// TwinCAT 3 PLC project benchmark
// ProgramVersion: 3.1.4026.13
// libraries:
//   Struckig, * (Stefan Besler)
//   Tc2_Standard, * (Beckhoff Automation GmbH)
//   Tc2_System, * (Beckhoff Automation GmbH)
//   Tc2_Utilities, * (Beckhoff Automation GmbH)
//   Tc3_Module, * (Beckhoff Automation GmbH)
// project tree:
//   / PlcTask.TcTTO
//   POUs/ MAIN.TcPOU
//   POUs/MovingStatistic/ MovingStatistic.TcPOU
//   POUs/Randomizer/ Randomizer.TcPOU
//   POUs/Random/ IRandom.TcIO, RandomGaussian.TcPOU, RandomUniform.TcPOU
//   POUs/Random/_Test/ RandomGaussianTest.TcPOU
// real-time tasks:
//   TASK PlcTask: cycle T#1ms, priority 1, ADS port 350

CONFIGURATION benchmark
    RESOURCE PLC ON TwinCAT3
        TASK PlcTask(INTERVAL := T#1ms, PRIORITY := 1);
        PROGRAM MAIN WITH PlcTask : MAIN;
    END_RESOURCE
END_CONFIGURATION

// ---- POUs/Random/IRandom.TcIO
INTERFACE IRandom

/// Returns the next random variable
METHOD Next : LREAL
END_METHOD

METHOD SetSeed
VAR_INPUT
  seed : INT;
END_VAR
END_METHOD

END_INTERFACE

// ---- POUs/MAIN.TcPOU
PROGRAM MAIN
VAR CONSTANT
  Dofs : ARRAY [0..3] OF SINT := [1, 3, 6, 7];
  IterationCount : INT := 5;
  TrajactoryCount : DINT := 64 * 1024;
END_VAR
VAR
  _positionDist : RandomGaussian(seed:=42, mu:=0, sigma:=4);
  _dynamicDist : RandomGaussian(seed:=43, mu:=0, sigma:=0.8);
  _limitDist : RandomUniform(seed:=44, lowerBound:=0, upperBound:=4);
  
  _p : Randomizer(_positionDist);
  _d : Randomizer(_dynamicDist);
  _l : Randomizer(_limitDist);
  
  _otg : Struckig.Otg(cycletime:=0.001, dofs:=0);
  
  _step : INT := 0;
  _dt, _it, _jt : DINT := 0;
  
  _trajectoryStatistic, _itStatistic, _worstStatistic : MovingStatistic;
  
  _averageMean, _worstMean, _averageSigma, _worstSigma : ARRAY[0..3] OF LREAL; 
  
  _cpucounter : Tc2_System.GETCPUACCOUNT;
END_VAR

REPEAT
  CASE _step
  OF
    // setup ****************************************************
    0: 
    // **********************************************************

      _otg.FB_init(TRUE, TRUE, 0.001, dofs:=Dofs[_dt]);
      _trajectoryStatistic.Reset();
      _itStatistic.Reset();
      _worstStatistic.Reset();
      
      _p.Fill(ADR(_otg.CurrentPosition), Dofs[_dt]);
      _p.Fill(ADR(_otg.TargetPosition), Dofs[_dt]);
      _l.FillMax(ADR(_otg.maxVelocity), Dofs[_dt], ADR(_otg.TargetVelocity));
      _l.FillMax(ADR(_otg.maxAcceleration), Dofs[_dt], ADR(_otg.TargetAcceleration));
      _l.Fill(ADR(_otg.maxJerk), Dofs[_dt]);
      CheckCalculation(_otg);  
    
      _step := 1;
  
    // iterate start ********************************************
    1: 
    // **********************************************************
    
      _trajectoryStatistic.Reset();
      _step := 2;
      
    // iterate loop *********************************************
    2: 
    // **********************************************************
    
      _p.Fill(ADR(_otg.CurrentPosition), Dofs[_dt]);
      _d.FillOrZero(ADR(_otg.CurrentVelocity), Dofs[_dt], 0.9);
      _d.FillOrZero(ADR(_otg.CurrentAcceleration), Dofs[_dt], 0.8);
      _p.Fill(ADR(_otg.TargetPosition), Dofs[_dt]);
      _d.FillOrZero(ADR(_otg.TargetVelocity), Dofs[_dt], 0.7);
      _d.FillOrZero(ADR(_otg.TargetAcceleration), Dofs[_dt], 0.6);
      _l.FillMax(ADR(_otg.MaxVelocity), Dofs[_dt], ADR(_otg.TargetVelocity));
      _l.FillMax(ADR(_otg.MaxAcceleration), Dofs[_dt], ADR(_otg.TargetAcceleration));
      _l.Fill(ADR(_otg.MaxJerk), Dofs[_dt]);
  
      IF NOT _otg.ValidateInput(FALSE, TRUE)
      THEN
        RETURN;
      END_IF
  
      _trajectoryStatistic.Append(CheckCalculation(_otg));
      _jt := _jt + 1;
      IF _jt > TrajactoryCount
      THEN
        _it := _it + 1;
        _jt := 0;        
        _step := 1;
        _itStatistic.Append(_trajectoryStatistic.Mean);
        _worstStatistic.Append(_trajectoryStatistic.Maximum);
      END_IF
      
      IF _it > IterationCount
      THEN
        _step := 3;
      END_IF
      
    // iterate end **********************************************
    3: 
    // **********************************************************

      _it := 0;
      _jt := 0;
      _averageMean[_dt] := _itStatistic.Mean;
      _averageSigma[_dt] := _itStatistic.Sigma;
      _worstMean[_dt] := _worstStatistic.Mean;
      _worstSigma[_dt] := _worstStatistic.Sigma;      
      _dt := _dt + 1;
      _step := SEL(_dt > 3, 0, 4);

    // done******* **********************************************
    4: 
    // **********************************************************
      ; 
  END_CASE
UNTIL _step = 4 
AND_THEN TRUE // wtf, fix this already Beckhoff - no breakpoints without an additional condition!!!! 
END_REPEAT

_step := 4;

METHOD CheckCalculation : LREAL;
VAR_INPUT
  otg : REFERENCE TO Struckig.Otg;
END_VAR
VAR
  cpuAccount : UDINT;
END_VAR
_cpucounter(cpuAccountDW => cpuAccount);
otg();
_cpucounter();
CheckCalculation := (_cpucounter.cpuAccountDW - cpuAccount) * 0.1; // us
END_METHOD

END_PROGRAM

// ---- POUs/Random/RandomGaussian.TcPOU
FUNCTION_BLOCK RandomGaussian IMPLEMENTS IRandom
VAR
  _mu : LREAL;
  _sigma : LREAL;    
  _rnd : Tc2_System.DRAND;
END_VAR

METHOD FB_init : BOOL
VAR_INPUT
	bInitRetains : BOOL; // if TRUE, the retain variables are initialized (warm start / cold start)
	bInCopyCode : BOOL;  // if TRUE, the instance afterwards gets moved into the copy code (online change)
  seed : INT;  
  mu : LREAL;
  sigma : LREAL;
END_VAR
SetSeed(seed);
SetMean(mu);
SetSigma(sigma);
END_METHOD

/// Implementation of the Box-Muller transform for normal distributed random
/// variables. There are much faster methods for doing this.
/// Implementation taken from [here](https://en.wikipedia.org/wiki/Box%E2%80%93Muller_transform)
METHOD Next : LREAL
VAR
  u1, u2 : LREAL;
END_VAR
VAR CONSTANT
  Pi : LREAL := 3.14159265358979323846;
END_VAR
//create two random numbers, make sure u1 is greater than epsilon
REPEAT
  _rnd(Num => u1);
  _rnd(Num => u2);  
UNTIL u1 > 1E-8 END_REPEAT

//compute z0 and z1
Next  := (_sigma * SQRT(-2.0 * LOG(u1))) * COS(2*Pi * u2) + _mu;

// we do not need the 2nd randomly distributed variable
// z1 := mag * SIN(2*Struckig.Constants.Pi  * u2) + mu;
END_METHOD

METHOD FINAL SetMean
VAR_INPUT
  mu : LREAL;
END_VAR
_mu := mu;
END_METHOD

METHOD FINAL SetSeed
VAR_INPUT
  seed : INT;
END_VAR
_rnd.Seed := seed;
END_METHOD

METHOD FINAL SetSigma
VAR_INPUT
  sigma : LREAL;
END_VAR
_sigma := sigma;
END_METHOD

END_FUNCTION_BLOCK

// ---- POUs/Random/RandomUniform.TcPOU
FUNCTION_BLOCK RandomUniform IMPLEMENTS IRandom
VAR
  _lowerBound : LREAL;
  _upperBound : LREAL;  
  _rnd : Tc2_System.DRAND;
END_VAR

METHOD FB_init : BOOL
VAR_INPUT
	bInitRetains : BOOL; // if TRUE, the retain variables are initialized (warm start / cold start)
	bInCopyCode : BOOL;  // if TRUE, the instance afterwards gets moved into the copy code (online change)
  seed : INT;      
  lowerBound : LREAL;
  upperBound : LREAL;
END_VAR
SetSeed(seed);
SetBounds(lowerBound, upperBound);
END_METHOD

METHOD Next : LREAL
_rnd();
Next := _rnd.Num * (_upperBound-_lowerBound) + _lowerBound;
END_METHOD

METHOD FINAL SetBounds
VAR_INPUT
  lowerBound : LREAL;
  upperBound : LREAL;
END_VAR
_lowerBound := lowerBound;
_upperBound := upperBound;
END_METHOD

METHOD FINAL SetSeed
VAR_INPUT
  seed : INT;
END_VAR
_rnd.Seed := seed;
END_METHOD

END_FUNCTION_BLOCK

// ---- POUs/Randomizer/Randomizer.TcPOU
FUNCTION_BLOCK Randomizer
VAR
  _rndUniform : RandomUniform(seed:=0, lowerBound:=0, upperBound:=1);
  _rnd : IRandom;
END_VAR

METHOD FB_init : BOOL
VAR_INPUT
	bInitRetains : BOOL; // if TRUE, the retain variables are initialized (warm start / cold start)
	bInCopyCode : BOOL;  // if TRUE, the instance afterwards gets moved into the copy code (online change)
  rnd : IRandom;
END_VAR
_rnd := rnd;
END_METHOD

METHOD Fill
VAR_INPUT
  data : POINTER TO LREAL;
  size : INT;
END_VAR
VAR
  i : INT;
END_VAR
FOR i:=0 TO size-1
DO
  data[i] := _rnd.Next();
END_FOR
END_METHOD

METHOD FillMax
VAR_INPUT
  data : POINTER TO LREAL;
  size : INT;
  offset : POINTER TO LREAL;
END_VAR
VAR
  i : INT;
END_VAR
FOR i:=0 TO size-1
DO
  data[i] := _rnd.Next() + ABS(offset[i]);
END_FOR
END_METHOD

METHOD FillMin
VAR_INPUT
  data : POINTER TO LREAL;
  size : INT;
  offset : POINTER TO LREAL;
END_VAR
VAR
  i : INT;
END_VAR
FOR i:=0 TO size-1
DO
  data[i] := _rnd.Next() - ABS(offset[i]);
END_FOR
END_METHOD

METHOD FillOrZero
VAR_INPUT
  data : POINTER TO LREAL;
  size : INT;
  p : LREAL; // value between 0-1 to adjust the probability of "fill with random number" to "fill with zero". p = 0.9 means that 10% of values are filled with zero
END_VAR
VAR
  i : INT;
END_VAR
FOR i:=0 TO size-1
DO
  data[i] := SEL(_rndUniform.Next() < p, 0, _rnd.Next());
END_FOR
END_METHOD

END_FUNCTION_BLOCK

// ---- POUs/MovingStatistic/MovingStatistic.TcPOU
FUNCTION_BLOCK MovingStatistic
VAR_OUTPUT
  Mean : LREAL;
  Sigma : LREAL;
  Size : DINT;
  Maximum : LREAL;
  Minimum : LREAL;
END_VAR
VAR
  _meanMem : LREAL;
  _varianceSum : LREAL;
END_VAR

METHOD Append
VAR_INPUT
  value : LREAL;
END_VAR
Size := Size + 1;
_meanMem := Mean;
Mean := (Mean + (value - Mean) / DINT_TO_LREAL(Size)); 

IF Size > 1
THEN
  _varianceSum := _varianceSum + (value - Mean) * (value - _meanMem);
  Sigma := SQRT(_varianceSum / (DINT_TO_LREAL(Size) - 1.0));
END_IF

IF value < Minimum
THEN
  Minimum := value;
END_IF

IF value > Maximum
THEN
  Maximum := value;
END_IF
END_METHOD

METHOD FB_init : BOOL
VAR_INPUT
	bInitRetains : BOOL; // if TRUE, the retain variables are initialized (warm start / cold start)
	bInCopyCode : BOOL;  // if TRUE, the instance afterwards gets moved into the copy code (online change)
END_VAR
Reset();
END_METHOD

METHOD FINAL Reset
VAR_INPUT
END_VAR
Mean := 0;
Sigma := 0;
Size := 0;
Minimum := 1.7976931348623157E+308;
Maximum := -1.7976931348623157E+308;
_varianceSum := 0;
END_METHOD

END_FUNCTION_BLOCK

// ---- POUs/Random/_Test/RandomGaussianTest.TcPOU
FUNCTION_BLOCK RandomGaussianTest EXTENDS RandomGaussian

Test_Next();

METHOD FB_init : BOOL
VAR_INPUT
	bInitRetains : BOOL; // if TRUE, the retain variables are initialized (warm start / cold start)
	bInCopyCode : BOOL;  // if TRUE, the instance afterwards gets moved into the copy code (online change)
  seed : INT; // not used, set to 0
  mu : LREAL; // not used, set to 0
  sigma : LREAL; // not used, set to 0
END_VAR
SetSeed(0);
SetMean(50);
SetSigma(4);
END_METHOD

METHOD Test_Next
VAR_OUTPUT
  expected : INT;
  actual : INT;
  message : STRING;
END_VAR
VAR_INST
  vals : ARRAY[0..99] OF DINT;
  v : LREAL;
  i : INT;
END_VAR
// create random numbers
FOR i:=0 TO 5000
DO
  v := Next();
  vals[LREAL_TO_INT(v)] := vals[LREAL_TO_INT(v)] + 1;
  i := i+1;
END_FOR

// check if the mean got the most counts
actual := 0;
FOR i:=0 TO 99
DO
  IF vals[i] > vals[actual]
  THEN
    actual := i;
	END_IF
END_FOR

expected := 50;
message := 'The index with the most counts is not the mean value of the distribution';
END_METHOD

END_FUNCTION_BLOCK
